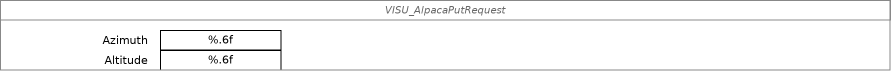
VISUALIZATION VISU_AlpacaPutSlewToAltAz  // 891x71
VAR_IN_OUT
	stInstance : ST_AlpacaPutSlewToAltAz;
END_VAR
    Frame (0,0 891x20)
        shows VISU_AlpacaPutRequest(stInstance := stInstance)
    Label (50,30 101x21), "Azimuth"
    Rectangle (160,30 121x20), "%.6f", text variable: stInstance.i_lrAzimuth
        OnMouseClick: write the text variable via Default
    Label (50,50 101x21), "Altitude"
    Rectangle (160,50 121x20), "%.6f", text variable: stInstance.i_lrAltitude
        OnMouseClick: write the text variable via Default
END_VISUALIZATION

(* stored: Version 1.1.0.1, ProductVersion 3.1.4024.12
   Visu VISU_AlpacaPutSlewToAltAz: Id {96f25ff3-6f48-4082-93d4-914715f44662} *)
